// TIA Portal V18 export
DATA_BLOCK "AutoProcessData_Buffer"   // DB1601
{ S7_Optimized_Access := 'FALSE' }
// stored: AutoNumber false
   VAR RETAIN
      DataBuffer : Array[0..55] of "ProcessDatad";
      DataBuffer_1 : "ProcessDatad";
      DataBuffer_2 { S7_SetPoint := 'True'} : "ProcessDatad";
      DataBuffer_3 { S7_SetPoint := 'True'} : "ProcessDatad";
      DataBuffer_4 { S7_SetPoint := 'True'} : "ProcessDatad";
      DataBuffer_5 { S7_SetPoint := 'True'} : "ProcessDatad";
      DataBuffer_6 { S7_SetPoint := 'True'} : "ProcessDatad";
      VAL { S7_SetPoint := 'True'} : Int;
      SelectButton : Int;
      Button_2 : Bool;
      Button_3 : Bool;
      Button_4 : Bool;
      Button_5 : Bool;
      Button_6 : Bool;
   END_VAR
BEGIN
END_DATA_BLOCK
